# EPICS substitutions: pearlJawsApp/Db/pearljawset.substitutions
global {P=\$(P), MOD_TO_SAMPLE=\$(MOD_TO_SAMPLE)}

file "$(TOP)/jawsManagerApp/Db/common.template" {
	{DIR=H, INIT_MOD_GAP=\$(MOD_GAP_WIDTH), EGU="mm"}
	{DIR=V, INIT_MOD_GAP=\$(MOD_GAP_HEIGHT), EGU="mm"}
}

file "$(TOP)/jawsManagerApp/Db/jaws_manager_single.template" {
    {JAW="JAWS1", MOD_TO_JAW="\$(MOD_TO_JAWS1)"}
    {JAW="JAWS2", MOD_TO_JAW="\$(MOD_TO_JAWS2)"}
    {JAW="JAWS3", MOD_TO_JAW="\$(MOD_TO_JAWS3)"}
}
